// TIA Portal V18 export
DATA_BLOCK "HSC_variables"   // DB2
{ S7_Optimized_Access := 'TRUE' }
VERSION : 0.1
// stored: AutoNumber true, IsOnlyStoredInLoadMemory false, IsRetainMemResEnabled false, IsWriteProtectedInAS false, MemoryReserve 100
   VAR
      timer_drain_time : Time := T#2s;
   END_VAR
BEGIN
END_DATA_BLOCK
